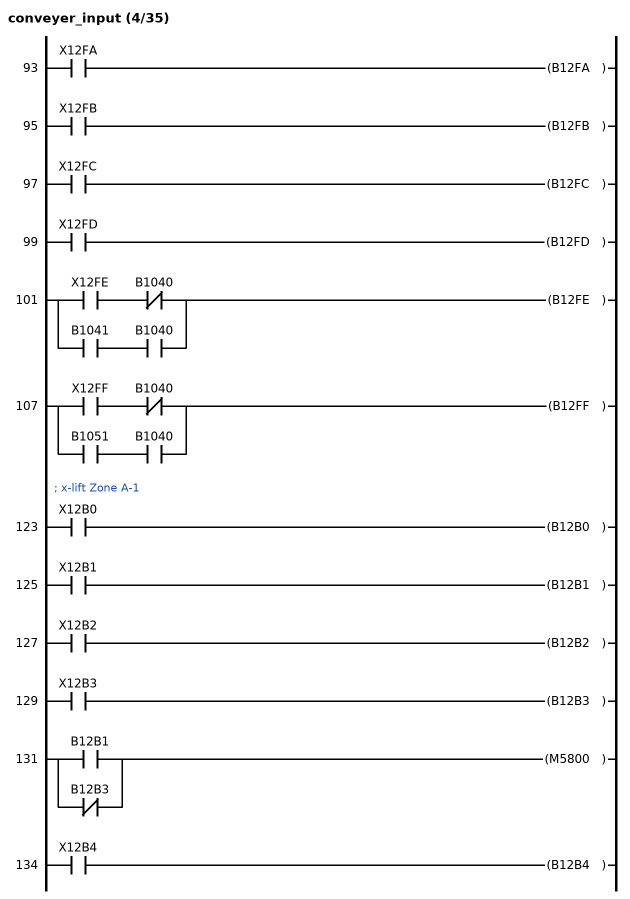
[picture p96: ladder of conveyer_input, rungs at steps 93 to 134]
93    LD      X12FA
      OUT     B12FA
95    LD      X12FB
      OUT     B12FB
97    LD      X12FC
      OUT     B12FC
99    LD      X12FD
      OUT     B12FD
101   LD      X12FE
      ANI     B1040
      LD      B1041
      AND     B1040
      ORB
      OUT     B12FE
107   LD      X12FF
      ANI     B1040
      LD      B1051
      AND     B1040
      ORB
      OUT     B12FF
; x-lift Zone A-1
123   LD      X12B0
      OUT     B12B0
125   LD      X12B1
      OUT     B12B1
127   LD      X12B2
      OUT     B12B2
129   LD      X12B3
      OUT     B12B3
131   LD      B12B1
      ORI     B12B3
      OUT     M5800
134   LD      X12B4
      OUT     B12B4
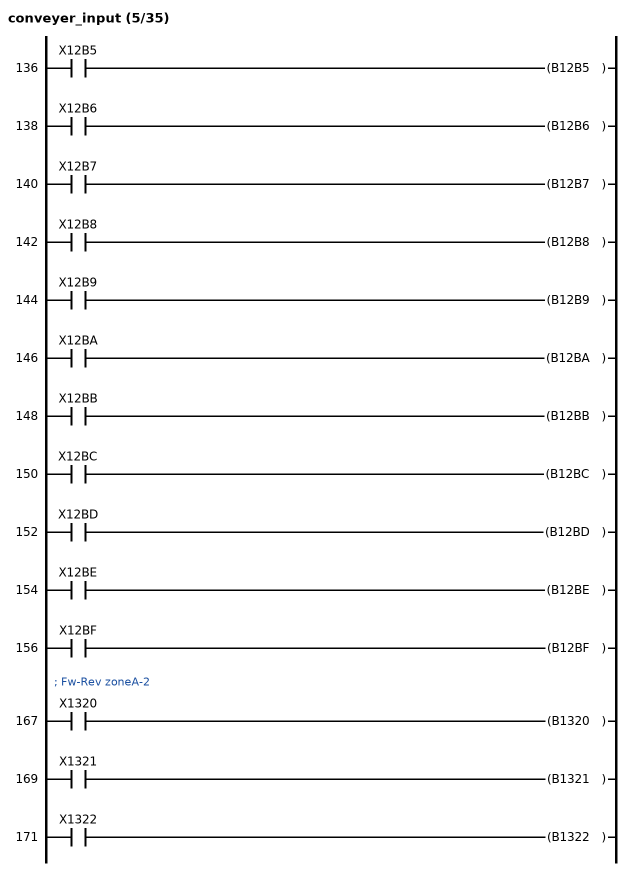
136   LD      X12B5
      OUT     B12B5
138   LD      X12B6
      OUT     B12B6
140   LD      X12B7
      OUT     B12B7
142   LD      X12B8
      OUT     B12B8
144   LD      X12B9
      OUT     B12B9
146   LD      X12BA
      OUT     B12BA
148   LD      X12BB
      OUT     B12BB
150   LD      X12BC
      OUT     B12BC
152   LD      X12BD
      OUT     B12BD
154   LD      X12BE
      OUT     B12BE
156   LD      X12BF
      OUT     B12BF
; Fw-Rev zoneA-2
167   LD      X1320
      OUT     B1320
169   LD      X1321
      OUT     B1321
171   LD      X1322
      OUT     B1322
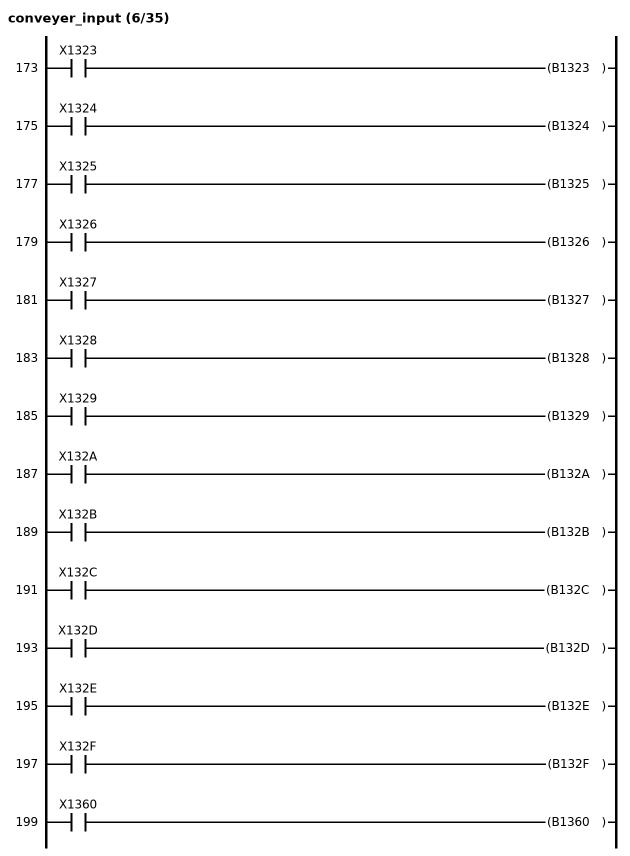
173   LD      X1323
      OUT     B1323
175   LD      X1324
      OUT     B1324
177   LD      X1325
      OUT     B1325
179   LD      X1326
      OUT     B1326
181   LD      X1327
      OUT     B1327
183   LD      X1328
      OUT     B1328
185   LD      X1329
      OUT     B1329
187   LD      X132A
      OUT     B132A
189   LD      X132B
      OUT     B132B
191   LD      X132C
      OUT     B132C
193   LD      X132D
      OUT     B132D
195   LD      X132E
      OUT     B132E
197   LD      X132F
      OUT     B132F
199   LD      X1360
      OUT     B1360
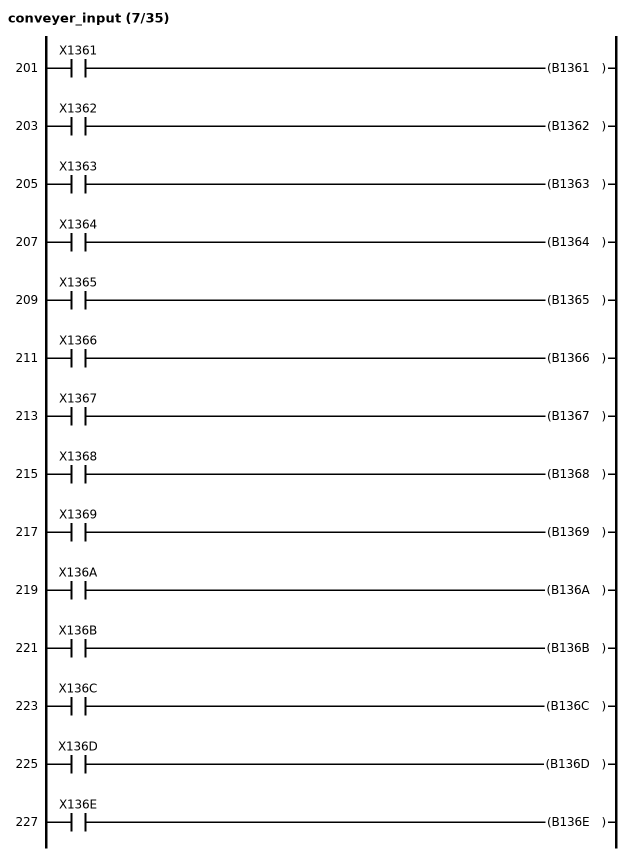
201   LD      X1361
      OUT     B1361
203   LD      X1362
      OUT     B1362
205   LD      X1363
      OUT     B1363
207   LD      X1364
      OUT     B1364
209   LD      X1365
      OUT     B1365
211   LD      X1366
      OUT     B1366
213   LD      X1367
      OUT     B1367
215   LD      X1368
      OUT     B1368
217   LD      X1369
      OUT     B1369
219   LD      X136A
      OUT     B136A
221   LD      X136B
      OUT     B136B
223   LD      X136C
      OUT     B136C
225   LD      X136D
      OUT     B136D
227   LD      X136E
      OUT     B136E
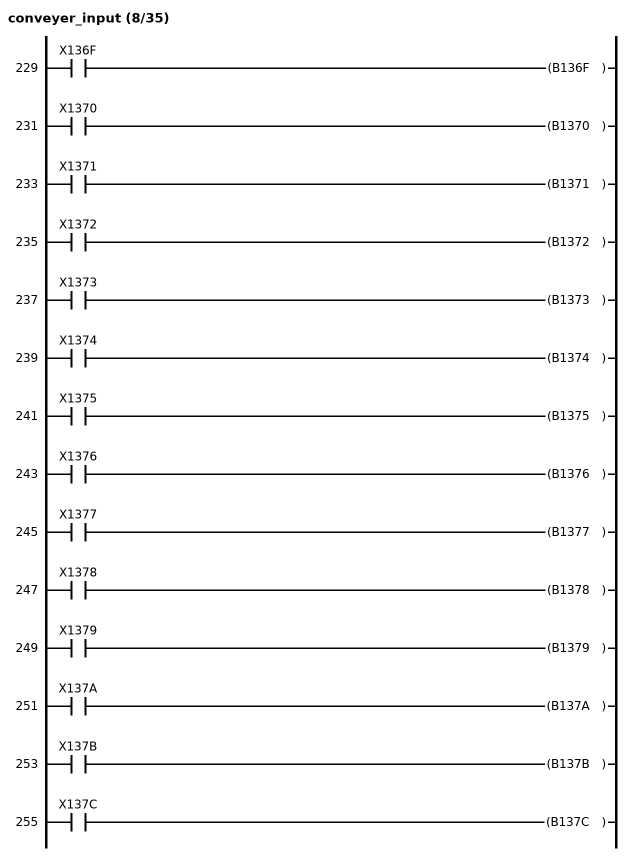
229   LD      X136F
      OUT     B136F
231   LD      X1370
      OUT     B1370
233   LD      X1371
      OUT     B1371
235   LD      X1372
      OUT     B1372
237   LD      X1373
      OUT     B1373
239   LD      X1374
      OUT     B1374
241   LD      X1375
      OUT     B1375
243   LD      X1376
      OUT     B1376
245   LD      X1377
      OUT     B1377
247   LD      X1378
      OUT     B1378
249   LD      X1379
      OUT     B1379
251   LD      X137A
      OUT     B137A
253   LD      X137B
      OUT     B137B
255   LD      X137C
      OUT     B137C
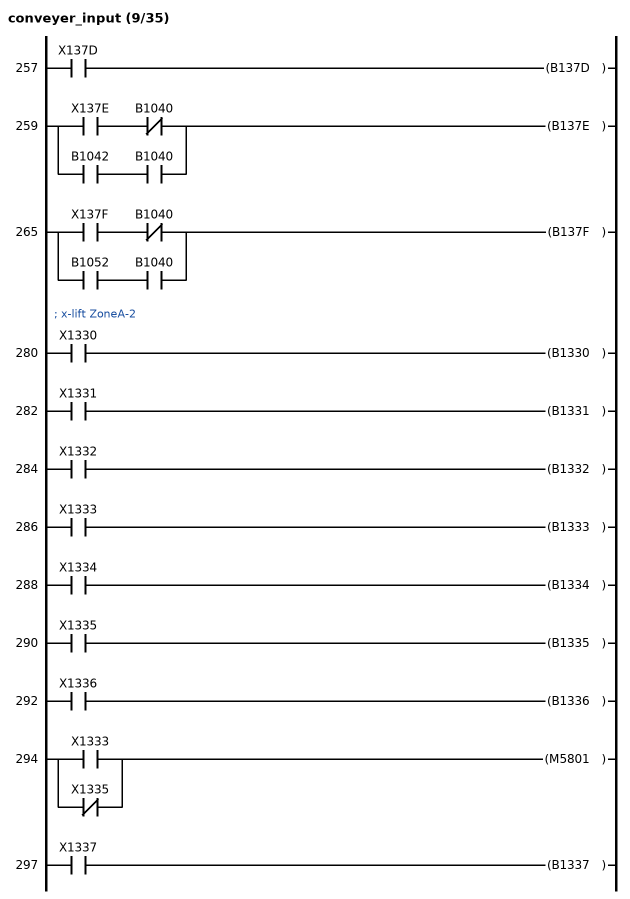
257   LD      X137D
      OUT     B137D
259   LD      X137E
      ANI     B1040
      LD      B1042
      AND     B1040
      ORB
      OUT     B137E
265   LD      X137F
      ANI     B1040
      LD      B1052
      AND     B1040
      ORB
      OUT     B137F
; x-lift ZoneA-2
280   LD      X1330
      OUT     B1330
282   LD      X1331
      OUT     B1331
284   LD      X1332
      OUT     B1332
286   LD      X1333
      OUT     B1333
288   LD      X1334
      OUT     B1334
290   LD      X1335
      OUT     B1335
292   LD      X1336
      OUT     B1336
294   LD      X1333
      ORI     X1335
      OUT     M5801
297   LD      X1337
      OUT     B1337
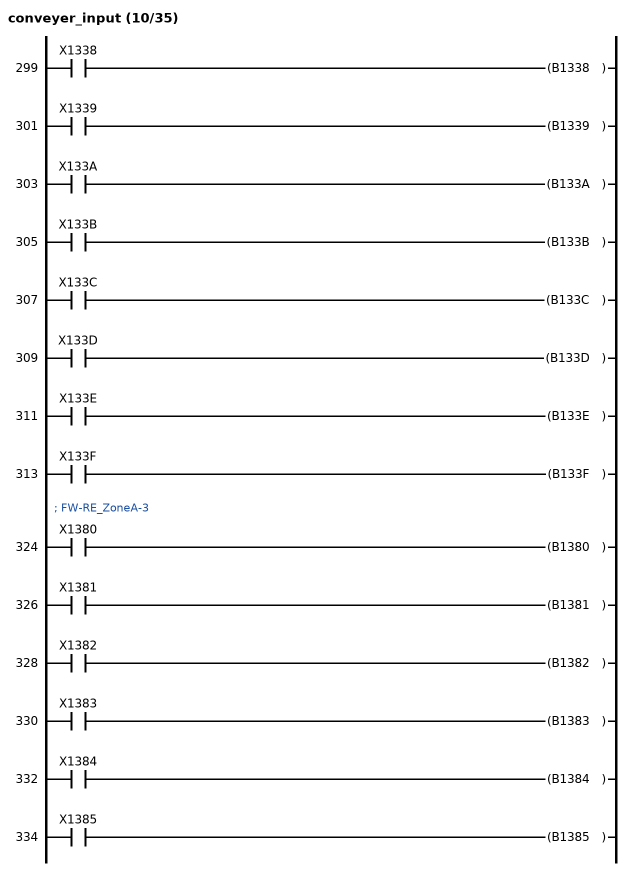
299   LD      X1338
      OUT     B1338
301   LD      X1339
      OUT     B1339
303   LD      X133A
      OUT     B133A
305   LD      X133B
      OUT     B133B
307   LD      X133C
      OUT     B133C
309   LD      X133D
      OUT     B133D
311   LD      X133E
      OUT     B133E
313   LD      X133F
      OUT     B133F
; FW-RE_ZoneA-3
324   LD      X1380
      OUT     B1380
326   LD      X1381
      OUT     B1381
328   LD      X1382
      OUT     B1382
330   LD      X1383
      OUT     B1383
332   LD      X1384
      OUT     B1384
334   LD      X1385
      OUT     B1385
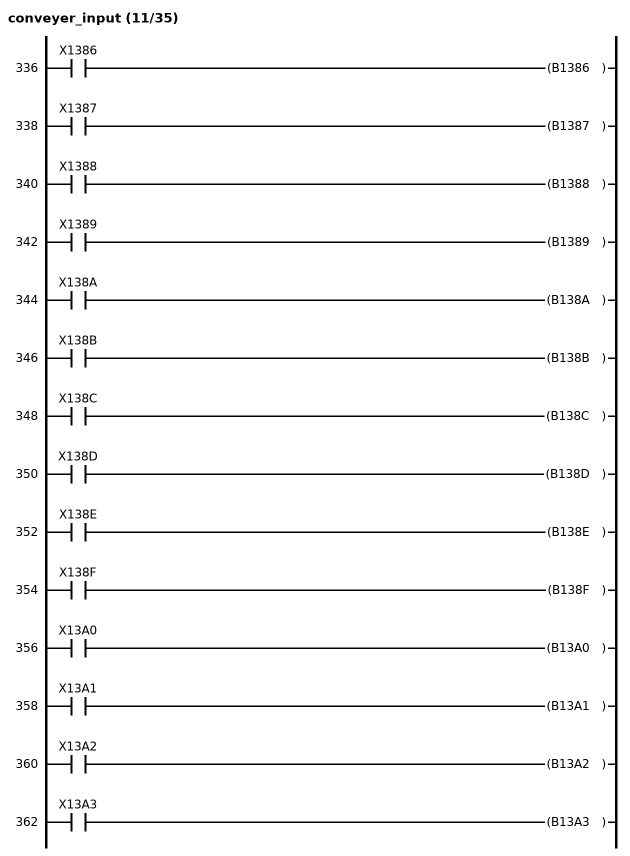
336   LD      X1386
      OUT     B1386
338   LD      X1387
      OUT     B1387
340   LD      X1388
      OUT     B1388
342   LD      X1389
      OUT     B1389
344   LD      X138A
      OUT     B138A
346   LD      X138B
      OUT     B138B
348   LD      X138C
      OUT     B138C
350   LD      X138D
      OUT     B138D
352   LD      X138E
      OUT     B138E
354   LD      X138F
      OUT     B138F
356   LD      X13A0
      OUT     B13A0
358   LD      X13A1
      OUT     B13A1
360   LD      X13A2
      OUT     B13A2
362   LD      X13A3
      OUT     B13A3
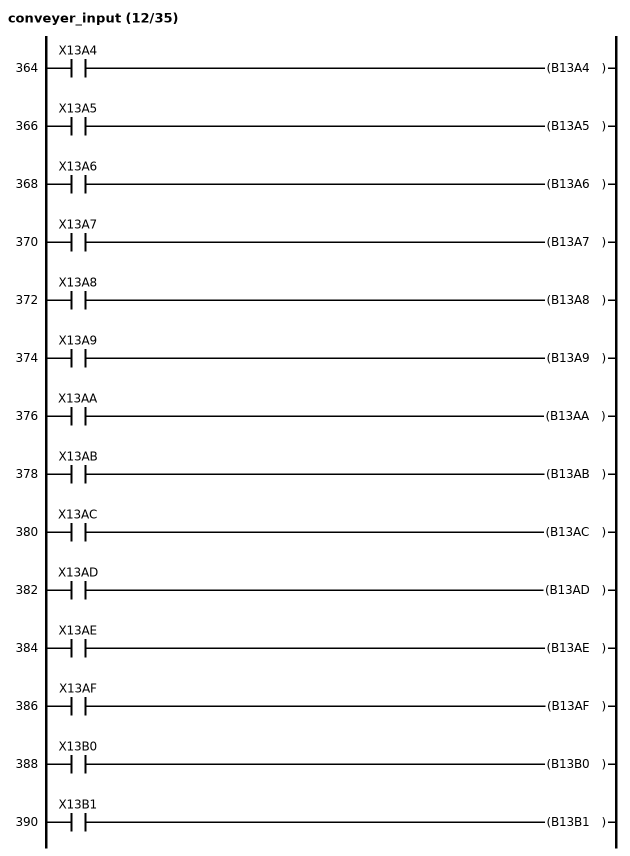
364   LD      X13A4
      OUT     B13A4
366   LD      X13A5
      OUT     B13A5
368   LD      X13A6
      OUT     B13A6
370   LD      X13A7
      OUT     B13A7
372   LD      X13A8
      OUT     B13A8
374   LD      X13A9
      OUT     B13A9
376   LD      X13AA
      OUT     B13AA
378   LD      X13AB
      OUT     B13AB
380   LD      X13AC
      OUT     B13AC
382   LD      X13AD
      OUT     B13AD
384   LD      X13AE
      OUT     B13AE
386   LD      X13AF
      OUT     B13AF
388   LD      X13B0
      OUT     B13B0
390   LD      X13B1
      OUT     B13B1
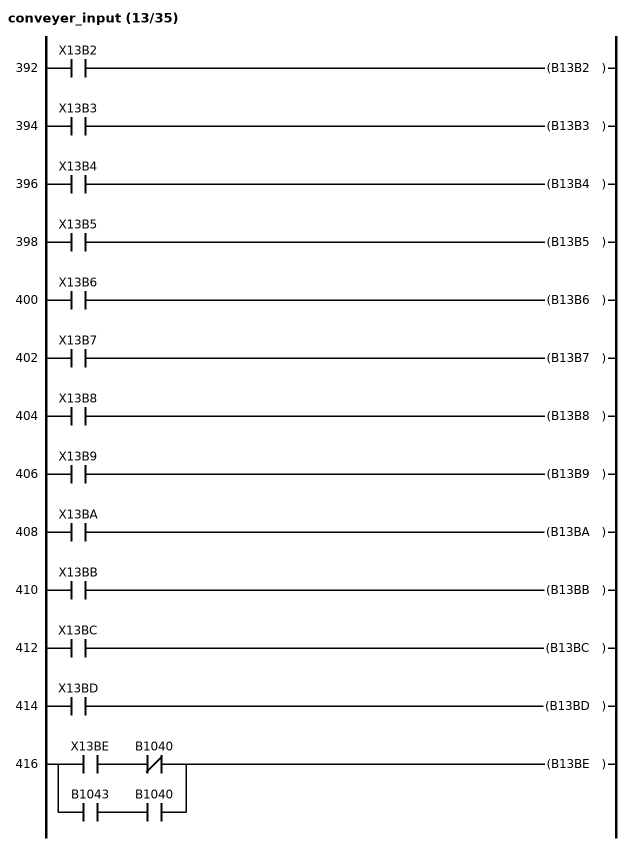
392   LD      X13B2
      OUT     B13B2
394   LD      X13B3
      OUT     B13B3
396   LD      X13B4
      OUT     B13B4
398   LD      X13B5
      OUT     B13B5
400   LD      X13B6
      OUT     B13B6
402   LD      X13B7
      OUT     B13B7
404   LD      X13B8
      OUT     B13B8
406   LD      X13B9
      OUT     B13B9
408   LD      X13BA
      OUT     B13BA
410   LD      X13BB
      OUT     B13BB
412   LD      X13BC
      OUT     B13BC
414   LD      X13BD
      OUT     B13BD
416   LD      X13BE
      ANI     B1040
      LD      B1043
      AND     B1040
      ORB
      OUT     B13BE
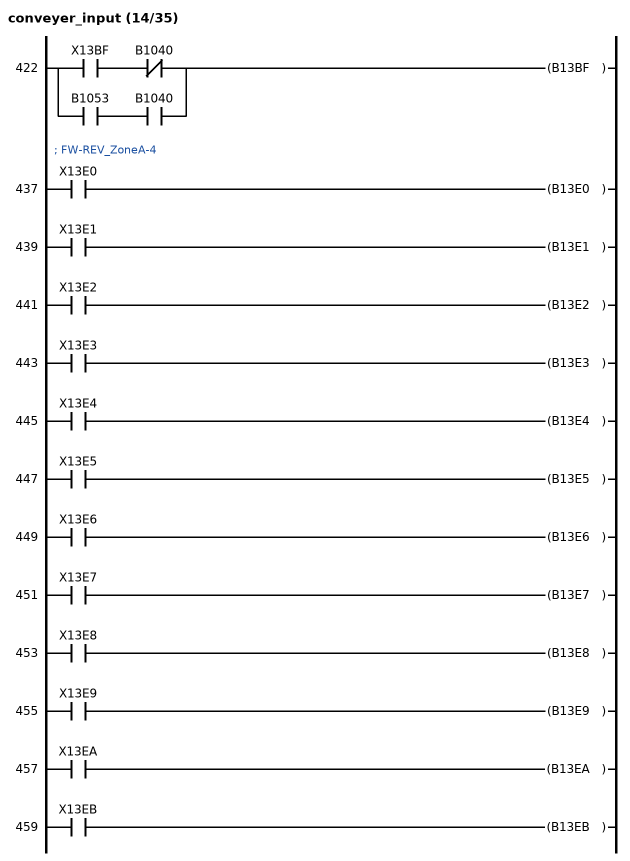
422   LD      X13BF
      ANI     B1040
      LD      B1053
      AND     B1040
      ORB
      OUT     B13BF
; FW-REV_ZoneA-4
437   LD      X13E0
      OUT     B13E0
439   LD      X13E1
      OUT     B13E1
441   LD      X13E2
      OUT     B13E2
443   LD      X13E3
      OUT     B13E3
445   LD      X13E4
      OUT     B13E4
447   LD      X13E5
      OUT     B13E5
449   LD      X13E6
      OUT     B13E6
451   LD      X13E7
      OUT     B13E7
453   LD      X13E8
      OUT     B13E8
455   LD      X13E9
      OUT     B13E9
457   LD      X13EA
      OUT     B13EA
459   LD      X13EB
      OUT     B13EB
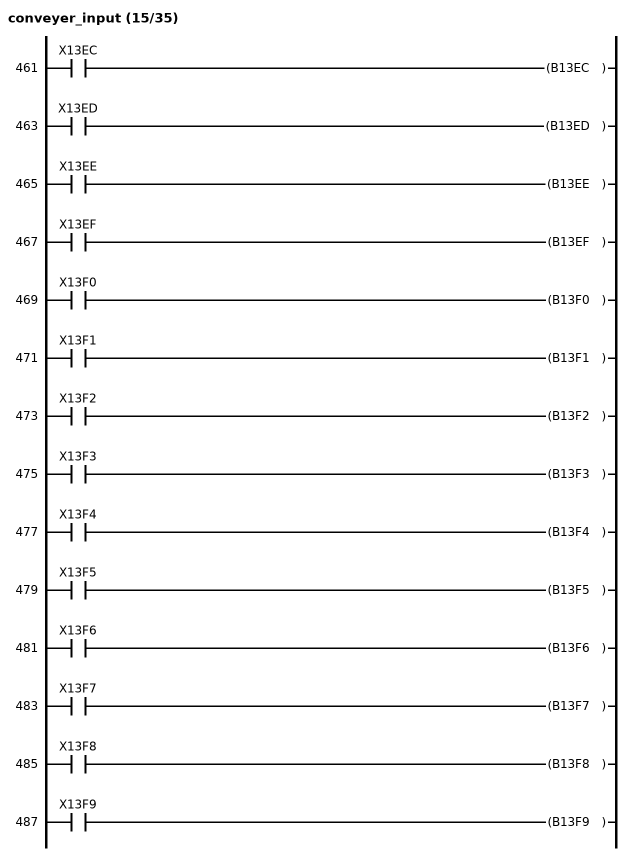
461   LD      X13EC
      OUT     B13EC
463   LD      X13ED
      OUT     B13ED
465   LD      X13EE
      OUT     B13EE
467   LD      X13EF
      OUT     B13EF
469   LD      X13F0
      OUT     B13F0
471   LD      X13F1
      OUT     B13F1
473   LD      X13F2
      OUT     B13F2
475   LD      X13F3
      OUT     B13F3
477   LD      X13F4
      OUT     B13F4
479   LD      X13F5
      OUT     B13F5
481   LD      X13F6
      OUT     B13F6
483   LD      X13F7
      OUT     B13F7
485   LD      X13F8
      OUT     B13F8
487   LD      X13F9
      OUT     B13F9
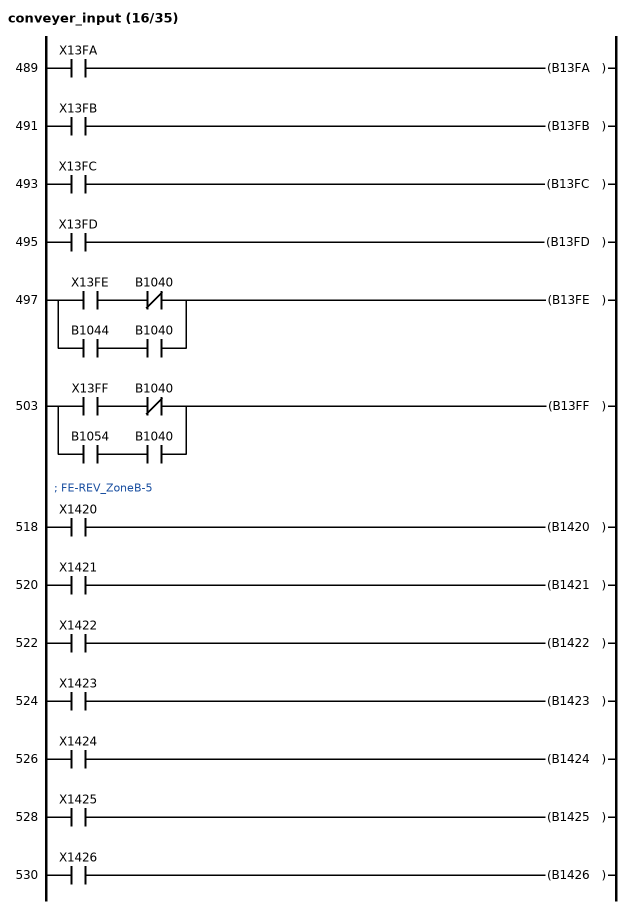
489   LD      X13FA
      OUT     B13FA
491   LD      X13FB
      OUT     B13FB
493   LD      X13FC
      OUT     B13FC
495   LD      X13FD
      OUT     B13FD
497   LD      X13FE
      ANI     B1040
      LD      B1044
      AND     B1040
      ORB
      OUT     B13FE
503   LD      X13FF
      ANI     B1040
      LD      B1054
      AND     B1040
      ORB
      OUT     B13FF
; FE-REV_ZoneB-5
518   LD      X1420
      OUT     B1420
520   LD      X1421
      OUT     B1421
522   LD      X1422
      OUT     B1422
524   LD      X1423
      OUT     B1423
526   LD      X1424
      OUT     B1424
528   LD      X1425
      OUT     B1425
530   LD      X1426
      OUT     B1426
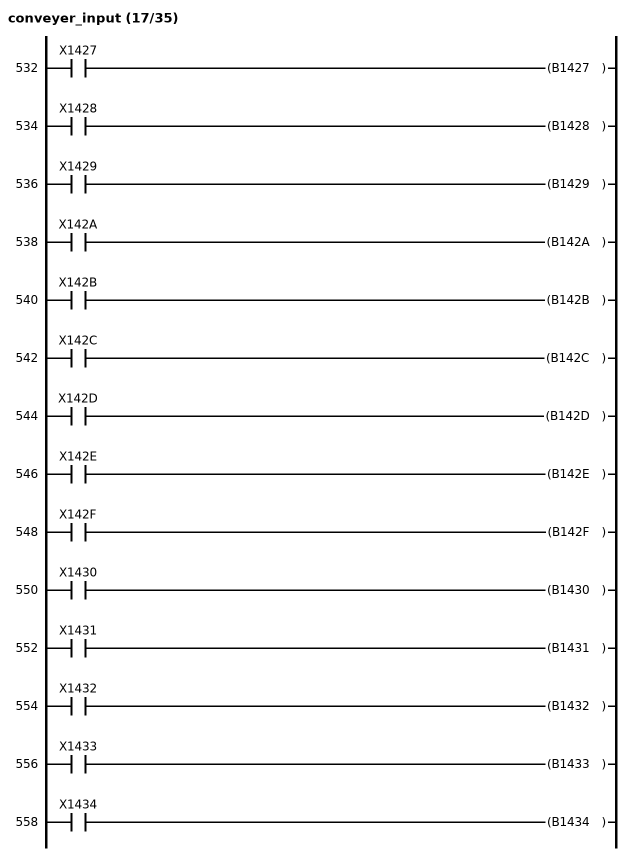
532   LD      X1427
      OUT     B1427
534   LD      X1428
      OUT     B1428
536   LD      X1429
      OUT     B1429
538   LD      X142A
      OUT     B142A
540   LD      X142B
      OUT     B142B
542   LD      X142C
      OUT     B142C
544   LD      X142D
      OUT     B142D
546   LD      X142E
      OUT     B142E
548   LD      X142F
      OUT     B142F
550   LD      X1430
      OUT     B1430
552   LD      X1431
      OUT     B1431
554   LD      X1432
      OUT     B1432
556   LD      X1433
      OUT     B1433
558   LD      X1434
      OUT     B1434
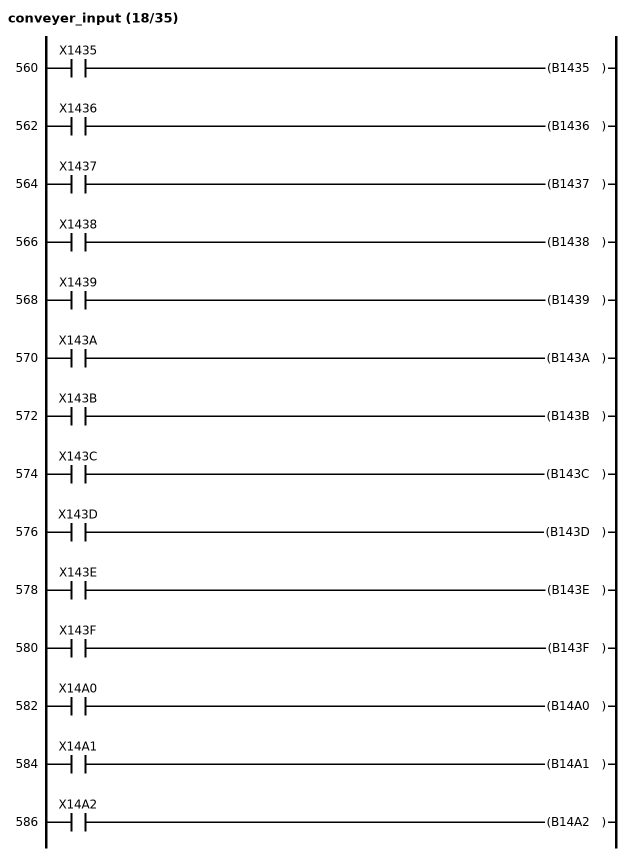
560   LD      X1435
      OUT     B1435
562   LD      X1436
      OUT     B1436
564   LD      X1437
      OUT     B1437
566   LD      X1438
      OUT     B1438
568   LD      X1439
      OUT     B1439
570   LD      X143A
      OUT     B143A
572   LD      X143B
      OUT     B143B
574   LD      X143C
      OUT     B143C
576   LD      X143D
      OUT     B143D
578   LD      X143E
      OUT     B143E
580   LD      X143F
      OUT     B143F
582   LD      X14A0
      OUT     B14A0
584   LD      X14A1
      OUT     B14A1
586   LD      X14A2
      OUT     B14A2
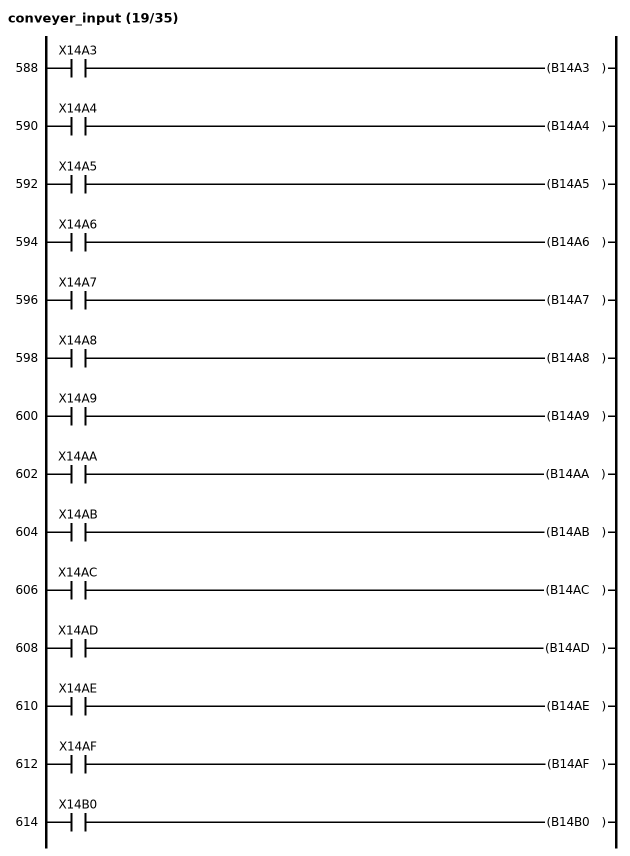
588   LD      X14A3
      OUT     B14A3
590   LD      X14A4
      OUT     B14A4
592   LD      X14A5
      OUT     B14A5
594   LD      X14A6
      OUT     B14A6
596   LD      X14A7
      OUT     B14A7
598   LD      X14A8
      OUT     B14A8
600   LD      X14A9
      OUT     B14A9
602   LD      X14AA
      OUT     B14AA
604   LD      X14AB
      OUT     B14AB
606   LD      X14AC
      OUT     B14AC
608   LD      X14AD
      OUT     B14AD
610   LD      X14AE
      OUT     B14AE
612   LD      X14AF
      OUT     B14AF
614   LD      X14B0
      OUT     B14B0
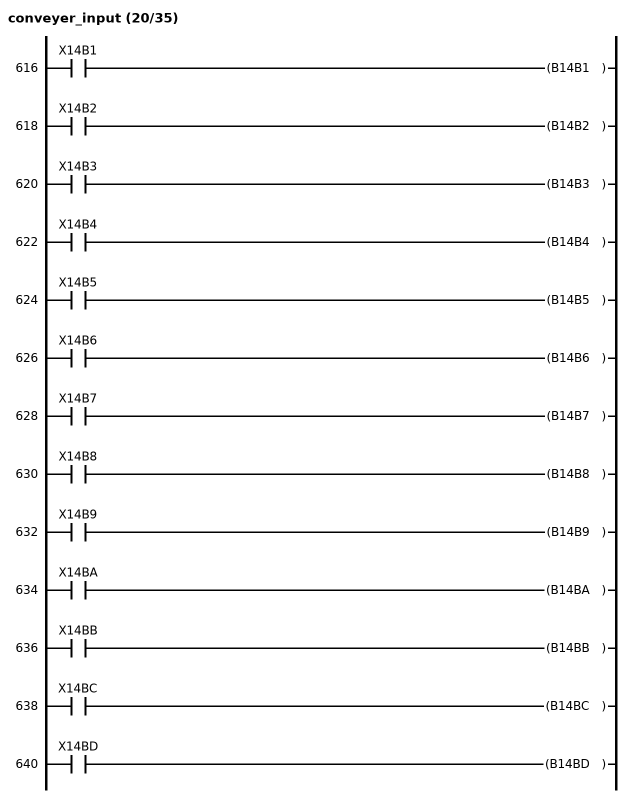
616   LD      X14B1
      OUT     B14B1
618   LD      X14B2
      OUT     B14B2
620   LD      X14B3
      OUT     B14B3
622   LD      X14B4
      OUT     B14B4
624   LD      X14B5
      OUT     B14B5
626   LD      X14B6
      OUT     B14B6
628   LD      X14B7
      OUT     B14B7
630   LD      X14B8
      OUT     B14B8
632   LD      X14B9
      OUT     B14B9
634   LD      X14BA
      OUT     B14BA
636   LD      X14BB
      OUT     B14BB
638   LD      X14BC
      OUT     B14BC
640   LD      X14BD
      OUT     B14BD
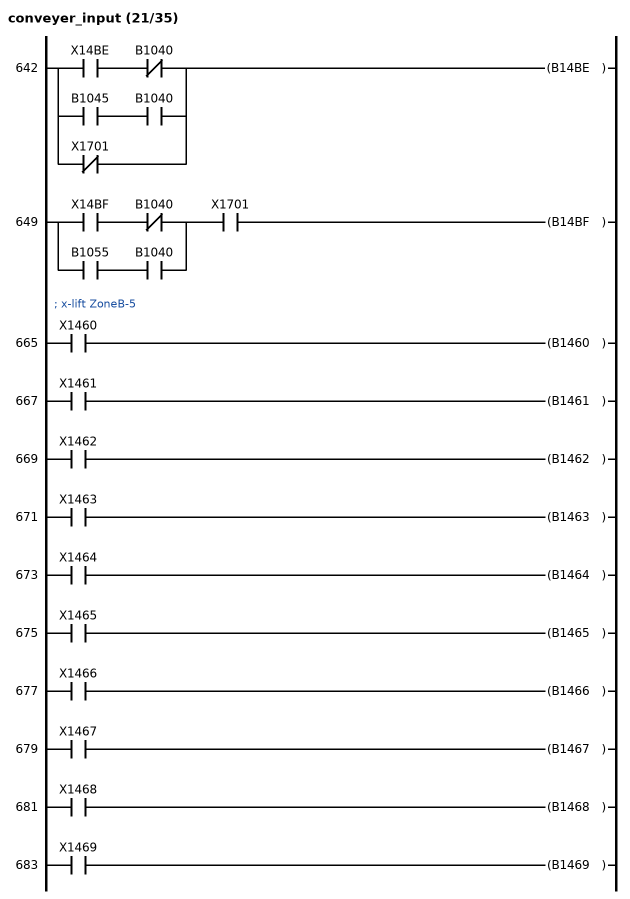
642   LD      X14BE
      ANI     B1040
      LD      B1045
      AND     B1040
      ORB
      ORI     X1701
      OUT     B14BE
649   LD      X14BF
      ANI     B1040
      LD      B1055
      AND     B1040
      ORB
      AND     X1701
      OUT     B14BF
; x-lift ZoneB-5
665   LD      X1460
      OUT     B1460
667   LD      X1461
      OUT     B1461
669   LD      X1462
      OUT     B1462
671   LD      X1463
      OUT     B1463
673   LD      X1464
      OUT     B1464
675   LD      X1465
      OUT     B1465
677   LD      X1466
      OUT     B1466
679   LD      X1467
      OUT     B1467
681   LD      X1468
      OUT     B1468
683   LD      X1469
      OUT     B1469
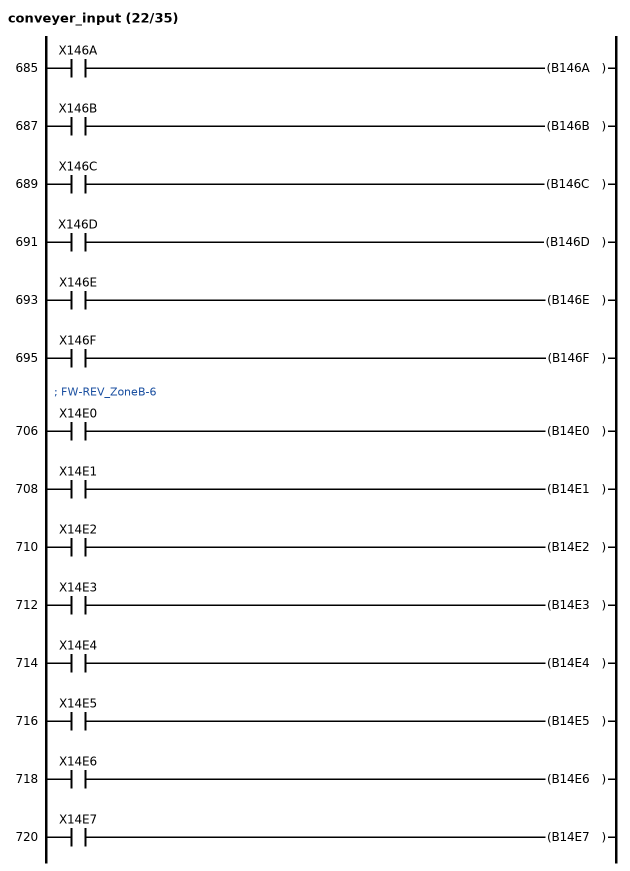
685   LD      X146A
      OUT     B146A
687   LD      X146B
      OUT     B146B
689   LD      X146C
      OUT     B146C
691   LD      X146D
      OUT     B146D
693   LD      X146E
      OUT     B146E
695   LD      X146F
      OUT     B146F
; FW-REV_ZoneB-6
706   LD      X14E0
      OUT     B14E0
708   LD      X14E1
      OUT     B14E1
710   LD      X14E2
      OUT     B14E2
712   LD      X14E3
      OUT     B14E3
714   LD      X14E4
      OUT     B14E4
716   LD      X14E5
      OUT     B14E5
718   LD      X14E6
      OUT     B14E6
720   LD      X14E7
      OUT     B14E7
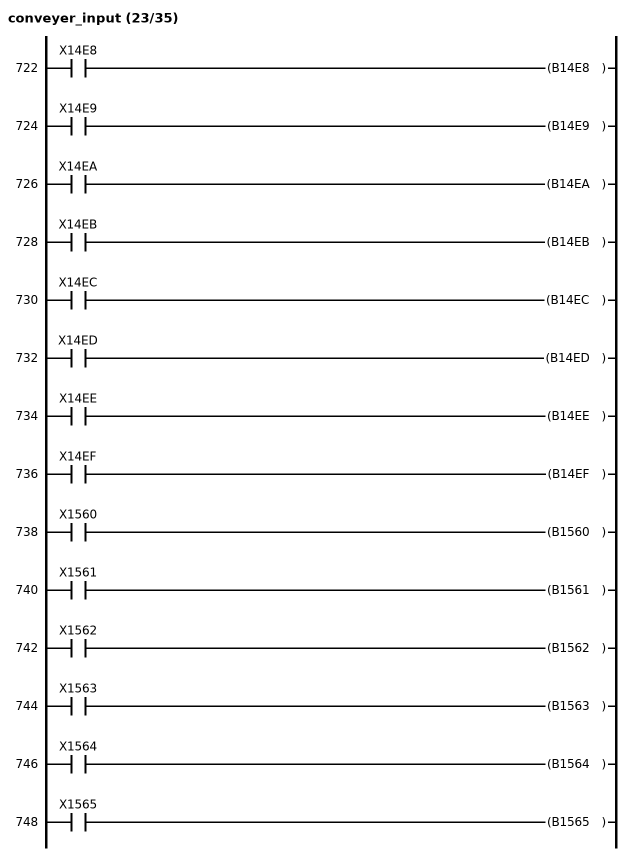
722   LD      X14E8
      OUT     B14E8
724   LD      X14E9
      OUT     B14E9
726   LD      X14EA
      OUT     B14EA
728   LD      X14EB
      OUT     B14EB
730   LD      X14EC
      OUT     B14EC
732   LD      X14ED
      OUT     B14ED
734   LD      X14EE
      OUT     B14EE
736   LD      X14EF
      OUT     B14EF
738   LD      X1560
      OUT     B1560
740   LD      X1561
      OUT     B1561
742   LD      X1562
      OUT     B1562
744   LD      X1563
      OUT     B1563
746   LD      X1564
      OUT     B1564
748   LD      X1565
      OUT     B1565
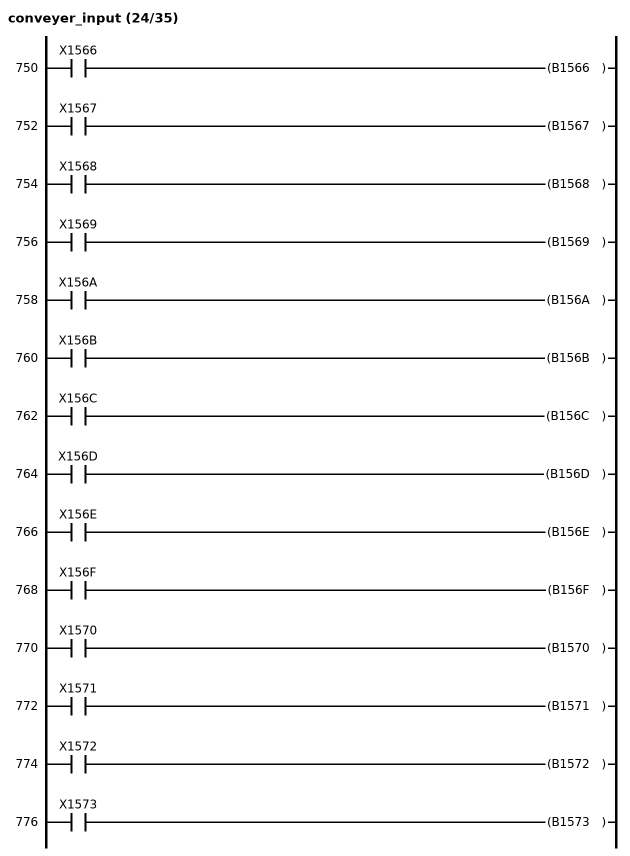
750   LD      X1566
      OUT     B1566
752   LD      X1567
      OUT     B1567
754   LD      X1568
      OUT     B1568
756   LD      X1569
      OUT     B1569
758   LD      X156A
      OUT     B156A
760   LD      X156B
      OUT     B156B
762   LD      X156C
      OUT     B156C
764   LD      X156D
      OUT     B156D
766   LD      X156E
      OUT     B156E
768   LD      X156F
      OUT     B156F
770   LD      X1570
      OUT     B1570
772   LD      X1571
      OUT     B1571
774   LD      X1572
      OUT     B1572
776   LD      X1573
      OUT     B1573
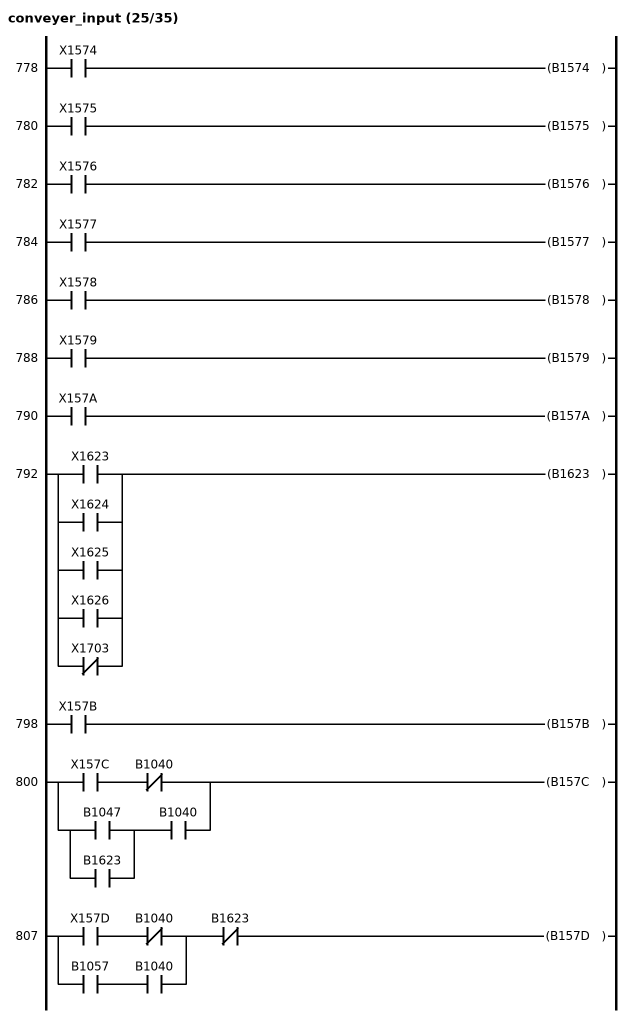
778   LD      X1574
      OUT     B1574
780   LD      X1575
      OUT     B1575
782   LD      X1576
      OUT     B1576
784   LD      X1577
      OUT     B1577
786   LD      X1578
      OUT     B1578
788   LD      X1579
      OUT     B1579
790   LD      X157A
      OUT     B157A
792   LD      X1623
      OR      X1624
      OR      X1625
      OR      X1626
      ORI     X1703
      OUT     B1623
798   LD      X157B
      OUT     B157B
800   LD      X157C
      ANI     B1040
      LD      B1047
      OR      B1623
      AND     B1040
      ORB
      OUT     B157C
807   LD      X157D
      ANI     B1040
      LD      B1057
      AND     B1040
      ORB
      ANI     B1623
      OUT     B157D
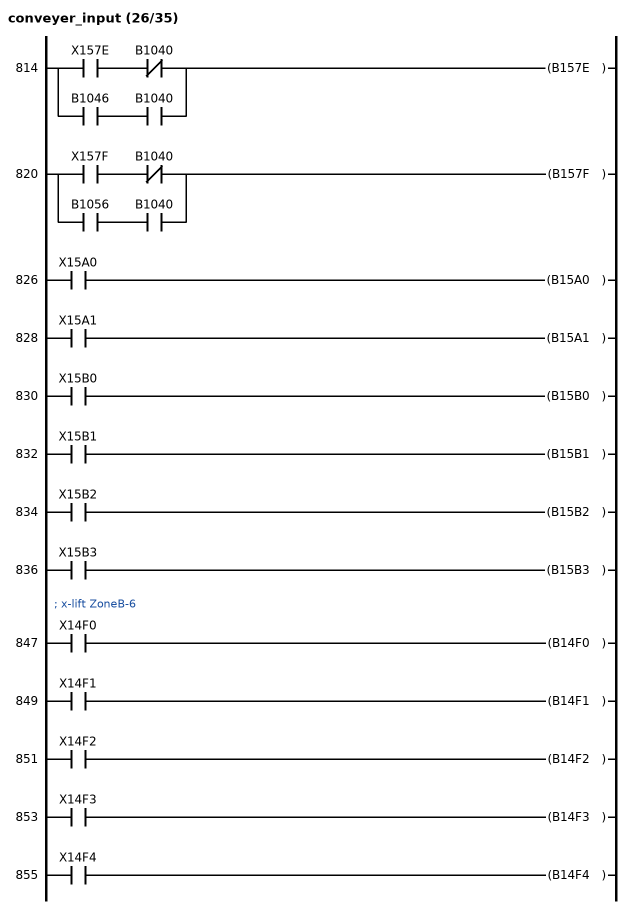
814   LD      X157E
      ANI     B1040
      LD      B1046
      AND     B1040
      ORB
      OUT     B157E
820   LD      X157F
      ANI     B1040
      LD      B1056
      AND     B1040
      ORB
      OUT     B157F
826   LD      X15A0
      OUT     B15A0
828   LD      X15A1
      OUT     B15A1
830   LD      X15B0
      OUT     B15B0
832   LD      X15B1
      OUT     B15B1
834   LD      X15B2
      OUT     B15B2
836   LD      X15B3
      OUT     B15B3
; x-lift ZoneB-6
847   LD      X14F0
      OUT     B14F0
849   LD      X14F1
      OUT     B14F1
851   LD      X14F2
      OUT     B14F2
853   LD      X14F3
      OUT     B14F3
855   LD      X14F4
      OUT     B14F4
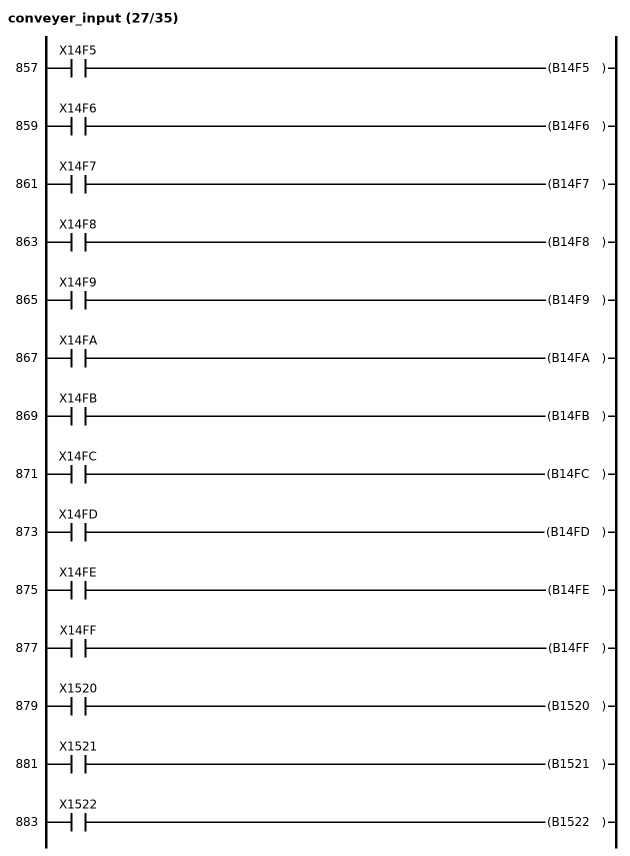
857   LD      X14F5
      OUT     B14F5
859   LD      X14F6
      OUT     B14F6
861   LD      X14F7
      OUT     B14F7
863   LD      X14F8
      OUT     B14F8
865   LD      X14F9
      OUT     B14F9
867   LD      X14FA
      OUT     B14FA
869   LD      X14FB
      OUT     B14FB
871   LD      X14FC
      OUT     B14FC
873   LD      X14FD
      OUT     B14FD
875   LD      X14FE
      OUT     B14FE
877   LD      X14FF
      OUT     B14FF
879   LD      X1520
      OUT     B1520
881   LD      X1521
      OUT     B1521
883   LD      X1522
      OUT     B1522
